TYPE T_CHM_Filename : T_MaxString;
END_TYPE

(* stored: Version 1.1.0.1, ProductVersion 3.1.4024.15
   DUT T_CHM_Filename: Id {d9cb45f6-1218-42f1-8f44-add809c0d405} *)
